TYPE ST_CoeParameterREAL :
STRUCT
	fValue : REAL;
	nIndex : WORD;
	nSubIndex : BYTE;
END_STRUCT
END_TYPE

(* stored: Version 1.1.0.1, ProductVersion 3.1.4022.18
   DUT ST_CoeParameterREAL: Id {32745d7c-8794-402c-bb36-b72b1589602b} *)
